// Mitsubishi GX Works2 project: GX W2 L2 Ex 1 DK c   PLC: FX3G

// global labels: Global1
VAR_GLOBAL
  iS1 AT X001 : BOOL;
  oLamp_1 AT Y001 : BOOL;
  oLamp_2 AT Y002 : BOOL;
END_VAR

// task Task_01 (event TRUE, interval 0, priority 31): POU_01

PROGRAM POU_01
VAR
  TON_1 : TON;
  TON_2 : TON;
END_VAR
(* structured ladder/FBD written out as ST: instructions are called as NAME(EN, inputs, outputs); _pN, _eN, _tN stand for wires *)
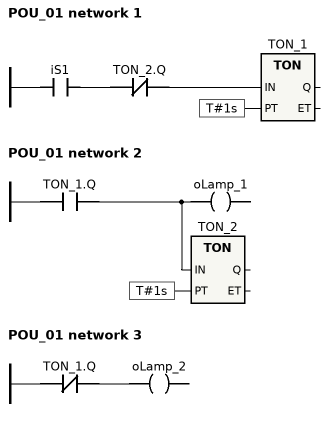
(* network 1 *)
TON_1(IN := iS1 AND NOT TON_2.Q, PT := T#1s);
(* network 2 *)
oLamp_1 := TON_1.Q;
TON_2(IN := TON_1.Q, PT := T#1s);
(* network 3 *)
oLamp_2 := NOT TON_1.Q;
END_PROGRAM
